PROGRAM ParallelPID
VAR
	prevError: REAL := 0;
	prevIntegral: REAL := 0;
END_VAR

END_PROGRAM

(* stored: Version 1.1.0.1, ProductVersion 3.1.4024.12
   POU ParallelPID: Id {c6bece98-9eca-4ec6-acee-eba02304d025}, SpecialFunc None *)
